// Library/POUs/Additional/MC_SoftSwitchTcp/Structures/SoftSwitchTcpOutCmd
{attribute 'pack_mode' := '1'} 
// ------------------------------------------------------------------------- 
//  SRCI Robot Library                                                
// ------------------------------------------------------------------------- 
//                                                                           
//  Object:      SoftSwitchTcpOutCmd                                       
//  Author:      Thorsten Brach                                                
//  Date:        2024-06-30
//
//  Description:                                              
//   
//                                                                           
//  Copyright: 
//    (C) 2024 Thorsten Brach. All rights reserved                                                                                                                                            
//             Licensed under the LGPL-3.0 license.
//                                                                           
//  Disclaimer:                                                                           
//    This project is provided without any guarantee and can be used for   
//    private and commercial purposes. Any use is at the user’s 
//    own risk and responsibility.
//
// -------------------------------------------------------------------------
TYPE SoftSwitchTcpOutCmd :
STRUCT
  /// If TRUE, the RA is in a compliant movement.
  SoftMovement : BOOL;
END_STRUCT
END_TYPE

// Library/POUs/Additional/MC_SoftSwitchTcp/Structures/SoftSwitchTcpParCmd
{attribute 'pack_mode' := '1'} 
// ------------------------------------------------------------------------- 
//  SRCI Robot Library                                                
// ------------------------------------------------------------------------- 
//                                                                           
//  Object:      SoftSwitchTcpParCmd                                       
//  Author:      Thorsten Brach                                                
//  Date:        2024-06-30
//
//  Description:                                              
//   
//                                                                           
//  Copyright: 
//    (C) 2024 Thorsten Brach. All rights reserved                                                                                                                                            
//             Licensed under the LGPL-3.0 license.
//                                                                           
//  Disclaimer:                                                                           
//    This project is provided without any guarantee and can be used for   
//    private and commercial purposes. Any use is at the user’s 
//    own risk and responsibility.
//
// -------------------------------------------------------------------------
TYPE SoftSwitchTcpParCmd :
STRUCT
  /// Defines type of reference coordinate system at which the robot can be moved in a compliant manner.
  ReferenceType       : ReferenceType;
  /// Index of tool or frame according to ReferenceType.
  /// • 0 (default): Flange/WS
  /// • 1..254: Tool/User frames
  ReferenceNo         : USINT;
  /// Relates to "LimitMode" with the setting "No limit defined". Defines for which cartesian axes the compliant motion is allowed. 
  /// If TRUE, the direction is enabled. Default value is FALSE. See Table 6-744 for bit assignment.
  CompliantAxes       : BYTE;
  /// Defines which parameters will limit the space, where the robot complies (at least one option must be supported)
  LimitMode           : LimitMode;
  /// Defines the type of the resistance force applied at the RA against the external force
  ResistanceForceMode : ResistanceForceMode;
  /// Relates to "ResistanceForceMode" with the setting "ResistanceForceTCP".
  /// Defines the resistance force level applied at the RA against the external force.
  /// • 0..99: Resistance is lower than robot vendor default. The lower the value, the easier the robot can be pushed away.
  /// • 100 (default): The value is aligned with the robot vendor-specific default value.
  /// • 101..200: Resistance is higher than robot vendor default. At maximum value "200" highest possible resistance against external force
  ResistanceForceTCP  : REAL;
  /// Relates to "ResistanceForceMode" with the setting "ResistanceForceAxis".
  /// Defines the resistance force level of the RA at the respective cartesian axis.
  ///  0..99: Resistance is lower than robot vendor default. The lower the value, the easier the robot can be pushed away.
  /// • 100 (default): The value is aligned with the robot vendor-specific default value.
  /// • 101..200: Resistance is higher than robot vendor default. At maximum value "200" highest possible resistance against external force.
  /// Index:
  /// • [0]: X-Axis O
  /// • [1]: Y-axis O
  /// • [2]: Z-axis O
  /// • [3]: RX-Direction O
  /// • [4]: RY-direction O
  /// • [5]: RZ-direction
  ResistanceForceAxis : ARRAY[0..5] OF REAL;
  /// Relates to "LimitMode" with the setting "Limit defined". 
  /// Limit values in the selected cartesian coordinate system (see input parameters ReferenceType and ReferenceNo).
  /// "0" is (default) the origin of the vector, the TCP position, at the start position of the robot.
  /// See Table 6-742 for the parameter index assignment.
  VectorData          : ARRAY[0..5] OF REAL;
END_STRUCT
END_TYPE

// Library/POUs/Additional/MC_SoftSwitchTcp/Structures/SoftSwitchTcpRecvData
{attribute 'pack_mode' := '1'} 
// ------------------------------------------------------------------------- 
//  SRCI Robot Library                                                
// ------------------------------------------------------------------------- 
//                                                                           
//  Object:      SoftSwitchTcpRecvData                                       
//  Author:      Thorsten Brach                                                
//  Date:        2024-06-30
//
//  Description:                                              
//   
//                                                                           
//  Copyright: 
//    (C) 2024 Thorsten Brach. All rights reserved                                                                                                                                            
//             Licensed under the LGPL-3.0 license.
//                                                                           
//  Disclaimer:                                                                           
//    This project is provided without any guarantee and can be used for   
//    private and commercial purposes. Any use is at the user’s 
//    own risk and responsibility.
//
// -------------------------------------------------------------------------
TYPE SoftSwitchTcpRecvData EXTENDS RspHeader :
STRUCT
  /// If TRUE, the RA is in a compliant movement.
  SoftMovement : BOOL;  
END_STRUCT
END_TYPE

// Library/POUs/Additional/MC_SoftSwitchTcp/Structures/SoftSwitchTcpSendData
{attribute 'pack_mode' := '1'}
// ------------------------------------------------------------------------- 
//  SRCI Robot Library                                                
// ------------------------------------------------------------------------- 
//                                                                           
//  Object:      SoftSwitchTcpSendData                                       
//  Author:      Thorsten Brach                                                
//  Date:        2024-06-30
//
//  Description:                                              
//   
//                                                                           
//  Copyright: 
//    (C) 2024 Thorsten Brach. All rights reserved                                                                                                                                            
//             Licensed under the LGPL-3.0 license.
//                                                                           
//  Disclaimer:                                                                           
//    This project is provided without any guarantee and can be used for   
//    private and commercial purposes. Any use is at the user’s 
//    own risk and responsibility.
//
// -------------------------------------------------------------------------
TYPE SoftSwitchTcpSendData EXTENDS CmdHeader: 
STRUCT
  /// Defines which parameters will limit the space, where the robot complies (at least one option must be supported)
  LimitMode           : LimitMode;
  /// Relates to "LimitMode" with the setting "No limit defined". Defines for which cartesian axes the compliant motion is allowed. 
  /// If TRUE, the direction is enabled. Default value is FALSE. See Table 6-744 for bit assignment.
  CompliantAxes       : BYTE;
  /// Defines type of reference coordinate system at which the robot can be moved in a compliant manner.
  ReferenceType       : ReferenceType;  
  /// Index of tool or frame according to ReferenceType.
  /// • 0 (default): Flange/WS
  /// • 1..254: Tool/User frames
  ReferenceNo         : USINT;
  /// Relates to "ResistanceForceMode" with the setting "ResistanceForceTCP".
  /// Defines the resistance force level applied at the RA against the external force.
  /// • 0..99: Resistance is lower than robot vendor default. The lower the value, the easier the robot can be pushed away.
  /// • 100 (default): The value is aligned with the robot vendor-specific default value.
  /// • 101..200: Resistance is higher than robot vendor default. At maximum value "200" highest possible resistance against external force
  ResistanceForceTCP  : INT;
  /// Relates to "ResistanceForceMode" with the setting "ResistanceForceAxis".
  /// Defines the resistance force level of the RA at the respective cartesian axis.
  ///  0..99: Resistance is lower than robot vendor default. The lower the value, the easier the robot can be pushed away.
  /// • 100 (default): The value is aligned with the robot vendor-specific default value.
  /// • 101..200: Resistance is higher than robot vendor default. At maximum value "200" highest possible resistance against external force.
  /// Index:
  /// • [0]: X-Axis O
  /// • [1]: Y-axis O
  /// • [2]: Z-axis O
  /// • [3]: RX-Direction O
  /// • [4]: RY-direction O
  /// • [5]: RZ-direction
  ResistanceForceAxis : ARRAY[0..5] OF UINT;
  /// Relates to "LimitMode" with the setting "Limit defined". 
  /// Limit values in the selected cartesian coordinate system (see input parameters ReferenceType and ReferenceNo).
  /// "0" is (default) the origin of the vector, the TCP position, at the start position of the robot.
  /// See Table 6-742 for the parameter index assignment.
  VectorData          : ARRAY[0..5] OF REAL;
  /// Defines the type of the resistance force applied at the RA against the external force
  ResistanceForceMode : ResistanceForceMode;
END_STRUCT
END_TYPE

// Library/POUs/Additional/MC_StopSubprogram/Structures/StopSubprogramOutCmd
{attribute 'pack_mode' := '1'} 
// ------------------------------------------------------------------------- 
//  SRCI Robot Library                                                
// ------------------------------------------------------------------------- 
//                                                                           
//  Object:      StopSubprogramOutCmd                                       
//  Author:      Thorsten Brach                                                
//  Date:        2024-08-01
//
//  Description:                                              
//   
//                                                                           
//  Copyright: 
//    (C) 2024 Thorsten Brach. All rights reserved                                                                                                                                            
//             Licensed under the LGPL-3.0 license.
//                                                                           
//  Disclaimer:                                                                           
//    This project is provided without any guarantee and can be used for   
//    private and commercial purposes. Any use is at the user’s 
//    own risk and responsibility.
//
// -------------------------------------------------------------------------
TYPE StopSubprogramOutCmd :
STRUCT
  OriginID           : INT;
  /// Relates to ListenerID >0
  /// Number of successful trigger -based command invocations
  /// For more information refer to chapter 5.5.12.4.
  InvocationCounter  : USINT;
END_STRUCT
END_TYPE

// Library/POUs/Additional/MC_StopSubprogram/Structures/StopSubprogramParCmd
{attribute 'pack_mode' := '1'} 
// ------------------------------------------------------------------------- 
//  SRCI Robot Library                                                
// ------------------------------------------------------------------------- 
//                                                                           
//  Object:      StopSubprogramParCmd                                       
//  Author:      Thorsten Brach                                                
//  Date:        2024-08-01
//
//  Description:                                              
//   
//                                                                           
//  Copyright: 
//    (C) 2024 Thorsten Brach. All rights reserved                                                                                                                                            
//             Licensed under the LGPL-3.0 license.
//                                                                           
//  Disclaimer:                                                                           
//    This project is provided without any guarantee and can be used for   
//    private and commercial purposes. Any use is at the user’s 
//    own risk and responsibility.
//
// -------------------------------------------------------------------------
TYPE StopSubprogramParCmd :
STRUCT
  /// Defines how target subprogram is defined
  StopMode          : StopMode;
  /// JobID or InstanceID of target subprogram according to selected StopMode
  /// • Refers to StopMode 0 (Stop via JobID) and 1 (Stop via InstanceID).
  /// • -1: Invalid (default)
  TargetID          : UINT;
  /// Defines the target sequence in which the command will be executed
  SequenceFlag      : SequenceFlag;
  /// ID of associated trigger function:
  /// • 0: No Trigger (default) - No trigger related behavior
  /// • >0: Triggero - Start executing when the trigger function with the identical EmitterID is triggered.
  /// Always positive.
  /// For more information, see chapter 5.5.12 Triggers
  ListenerID        : SINT;
  /// ID of Action that will be executed when this command is active
  /// • >0: Start Action - Start executing the Action function with the identical ListenerID.
  /// • <0: Stop Action  -  Stop executing the Action function with the identical ListenerID.
  /// • 0: No trigger (default)-  If no EmitterID is defined, the function will not trigger any Action during its execution
  /// For more information see section Triggers of this chapter or chapter 5.5.12.4.
  EmitterID          : ARRAY [0..3] OF SINT;  
END_STRUCT
END_TYPE

// Library/POUs/Additional/MC_StopSubprogram/Structures/StopSubprogramRecvData
{attribute 'pack_mode' := '1'} 
// ------------------------------------------------------------------------- 
//  SRCI Robot Library                                                
// ------------------------------------------------------------------------- 
//                                                                           
//  Object:      StopSubprogramRecvData                                       
//  Author:      Thorsten Brach                                                
//  Date:        2024-08-01
//
//  Description:                                              
//   
//                                                                           
//  Copyright: 
//    (C) 2024 Thorsten Brach. All rights reserved                                                                                                                                            
//             Licensed under the LGPL-3.0 license.
//                                                                           
//  Disclaimer:                                                                           
//    This project is provided without any guarantee and can be used for   
//    private and commercial purposes. Any use is at the user’s 
//    own risk and responsibility.
//
// -------------------------------------------------------------------------
TYPE StopSubprogramRecvData EXTENDS RspHeader :
STRUCT
  /// Relates to ListenerID >0
  /// Number of successful trigger-based command invocations - For more information refer TO chapter 5.5.12.4
  InvocationCounter : USINT;  
  /// Reserve
  Reserve           : SINT;
  /// Unique system-generated ID of the "Action" when the function is triggered.
  /// • >0: The "Action" is started by the trigger funcrion with identical FollowID.
  /// • <0: The "Action" is stopped by the trigger function with identical FollowID.
  /// For more information see chapter 5.5.12.4 EmitterID, ListenerID, FollowID and OriginID
  OriginID          : INT;
END_STRUCT
END_TYPE

// Library/POUs/Additional/MC_StopSubprogram/Structures/StopSubprogramSendData
{attribute 'pack_mode' := '1'}
// ------------------------------------------------------------------------- 
//  SRCI Robot Library                                                
// ------------------------------------------------------------------------- 
//                                                                           
//  Object:      StopSubprogramSendData                                       
//  Author:      Thorsten Brach                                                
//  Date:        2024-08-01
//
//  Description:                                              
//   
//                                                                           
//  Copyright: 
//    (C) 2024 Thorsten Brach. All rights reserved                                                                                                                                            
//             Licensed under the LGPL-3.0 license.
//                                                                           
//  Disclaimer:                                                                           
//    This project is provided without any guarantee and can be used for   
//    private and commercial purposes. Any use is at the user’s 
//    own risk and responsibility.
//
// -------------------------------------------------------------------------
TYPE StopSubprogramSendData EXTENDS CmdHeader: 
STRUCT
  /// ID of Action that will be executed when this command is active
  /// • >0: Start Action - Start executing the Action function with the identical ListenerID.
  /// • <0: Stop Action  -  Stop executing the Action function with the identical ListenerID.
  /// • 0: No trigger (default)-  If no EmitterID is defined, the function will not trigger any Action during its execution
  /// For more information see section Triggers of this chapter or chapter 5.5.12.4.
  EmitterID          : ARRAY [0..3] OF SINT;  
  /// ID of associated trigger function:
  /// • 0: No Trigger (default) - No trigger related behavior
  /// • >0: Triggero - Start executing when the trigger function with the identical EmitterID is triggered.
  /// Always positive.
  /// For more information, see chapter 5.5.12 Triggers
  ListenerID        : SINT;
  /// Reserve
  Reserve           : BYTE;
  /// JobID or InstanceID of target subprogram according to selected StopMode
  /// • Refers to StopMode 0 (Stop via JobID) and 1 (Stop via InstanceID).
  /// • -1: Invalid (default)
  TargetID          : UINT;
  /// Defines how target subprogram is defined
  StopMode          : USINT;  
END_STRUCT
END_TYPE

// Library/POUs/Additional/MC_UnitMeasurement/Structures/UnitMeasurementOutCmd
{attribute 'pack_mode' := '1'} 
// ------------------------------------------------------------------------- 
//  SRCI Robot Library                                                
// ------------------------------------------------------------------------- 
//                                                                           
//  Object:      UnitMeasurementOutCmd                                       
//  Author:      Thorsten Brach                                                
//  Date:        2024-06-30
//
//  Description:                                              
//   
//                                                                           
//  Copyright: 
//    (C) 2024 Thorsten Brach. All rights reserved                                                                                                                                            
//             Licensed under the LGPL-3.0 license.
//                                                                           
//  Disclaimer:                                                                           
//    This project is provided without any guarantee and can be used for   
//    private and commercial purposes. Any use is at the user’s 
//    own risk and responsibility.
//
// -------------------------------------------------------------------------
TYPE UnitMeasurementOutCmd :
STRUCT
  /// TRUE, while the measurement is active.
  MeasurementActive : BOOL;
  /// Measurement result depending on the measurement type setting of the "MeasuringMode".
  Result            : REAL;
  /// Unique system-generated ID of the "Action" when the function is triggered.
  /// • >0: The "Action" is started by the trigger function with identical FollowID.
  /// • <0: The "Action" is stopped by the trigger function with identical FollowID.
  /// For more information see chapter 5.5.12.4 EmitterID, ListenerID, FollowID and OriginID
  OriginID           : INT;
  /// Relates to ListenerID >0
  /// Number of successful trigger -based command invocations
  /// For more information refer to chapter 5.5.12.4.
  InvocationCounter  : USINT;
END_STRUCT
END_TYPE

// Library/POUs/Additional/MC_UnitMeasurement/Structures/UnitMeasurementParCmd
{attribute 'pack_mode' := '1'} 
// ------------------------------------------------------------------------- 
//  SRCI Robot Library                                                
// ------------------------------------------------------------------------- 
//                                                                           
//  Object:      UnitMeasurementParCmd                                       
//  Author:      Thorsten Brach                                                
//  Date:        2024-06-30
//
//  Description:                                              
//   
//                                                                           
//  Copyright: 
//    (C) 2024 Thorsten Brach. All rights reserved                                                                                                                                            
//             Licensed under the LGPL-3.0 license.
//                                                                           
//  Disclaimer:                                                                           
//    This project is provided without any guarantee and can be used for   
//    private and commercial purposes. Any use is at the user’s 
//    own risk and responsibility.
//
// -------------------------------------------------------------------------
TYPE UnitMeasurementParCmd :
STRUCT
  ///  Reaction type of measurement in relation to the trigger signal with the "ListenerID > 0" (at least one option must be supported):
  TriggerMode       : TriggerModeMeasurement;
  /// Relates to "TriggerMode" "No trigger related behavior".
  /// Set TRUE to start first measurement. Set TRUE again to receive new result data referring to previous rising edge of NewMeasurement.
  NewMeasurement    : BOOL;  
  /// Type of measurement (at least one option must be supported). 
 /// If the parameter is changed during the active measurement, the RC returns an error
  MeasuringMode     : MeasuringUnitMode;
  /// ID of the trigger function that may be triggered:
  /// • 0: Immediately (default). - Start executing THIS function immediately.
  /// • >0: Triggero Start executing when the trigger function with the identical EmitterID is called.
  /// For more information see chapter 5.5.12.4.
  ListenerID         : SINT;
END_STRUCT
END_TYPE

// Library/POUs/Additional/MC_UnitMeasurement/Structures/UnitMeasurementRecvData
{attribute 'pack_mode' := '1'} 
// ------------------------------------------------------------------------- 
//  SRCI Robot Library                                                
// ------------------------------------------------------------------------- 
//                                                                           
//  Object:      UnitMeasurementRecvData                                       
//  Author:      Thorsten Brach                                                
//  Date:        2024-06-30
//
//  Description:                                              
//   
//                                                                           
//  Copyright: 
//    (C) 2024 Thorsten Brach. All rights reserved                                                                                                                                            
//             Licensed under the LGPL-3.0 license.
//                                                                           
//  Disclaimer:                                                                           
//    This project is provided without any guarantee and can be used for   
//    private and commercial purposes. Any use is at the user’s 
//    own risk and responsibility.
//
// -------------------------------------------------------------------------
TYPE UnitMeasurementRecvData EXTENDS RspHeader :
STRUCT
  /// Relates to ListenerID >0
  /// Number of successful trigger -based command invocations
  /// For more information refer to chapter 5.5.12.4.
  InvocationCounter : USINT;
  /// Reserve
  Reserve           : SINT;
  /// Unique system-generated ID of the "Action" when the function is triggered.
  /// • >0: The "Action" is started by the trigger function with identical FollowID.
  /// • <0: The "Action" is stopped by the trigger function with identical FollowID.
  /// For more information see chapter 5.5.12.4 EmitterID, ListenerID, FollowID and OriginID
  OriginID          : INT;
  /// Measurement result depending on the measurement type setting of the "MeasuringMode".
  Result            : REAL;
  /// TRUE, while the measurement is active.
  MeasurementActive : BOOL;
  /// TRUE, when new result data was received from the RC.
  ResultNo          : USINT;
END_STRUCT
END_TYPE

// Library/POUs/Additional/MC_UnitMeasurement/Structures/UnitMeasurementSendData
{attribute 'pack_mode' := '1'}
// ------------------------------------------------------------------------- 
//  SRCI Robot Library                                                
// ------------------------------------------------------------------------- 
//                                                                           
//  Object:      UnitMeasurementSendData                                       
//  Author:      Thorsten Brach                                                
//  Date:        2024-06-30
//
//  Description:                                              
//   
//                                                                           
//  Copyright: 
//    (C) 2024 Thorsten Brach. All rights reserved                                                                                                                                            
//             Licensed under the LGPL-3.0 license.
//                                                                           
//  Disclaimer:                                                                           
//    This project is provided without any guarantee and can be used for   
//    private and commercial purposes. Any use is at the user’s 
//    own risk and responsibility.
//
// -------------------------------------------------------------------------
TYPE UnitMeasurementSendData EXTENDS CmdHeader: 
STRUCT
  EmitterID     : ARRAY [0..3] OF SINT;
  /// ID of the trigger function that may be triggered:
  /// • 0: Immediately (default). - Start executing THIS function immediately.
  /// • >0: Triggero Start executing when the trigger function with the identical EmitterID is called.
  /// For more information see chapter 5.5.12.4.
  ListenerID    : SINT;
  /// Reserve
  Reserve       : BYTE;
  ///  Reaction type of measurement in relation to the trigger signal with the "ListenerID > 0" (at least one option must be supported):
  TriggerMode   : TriggerModeMeasurement;
  /// Relates to "TriggerMode" "No trigger related behavior".
  /// Set TRUE to start first measurement. Set TRUE again to receive new result data referring to previous rising edge of NewMeasurement.
  MeasurementNo : USINT;
  /// Type of measurement (at least one option must be supported). 
  /// If the parameter is changed during the active measurement, the RC returns an error
  MeasuringMode : MeasuringUnitMode;


END_STRUCT
END_TYPE

// Library/POUs/Additional/MC_WriteCallSubprogramCyclic/Structures/WriteCallSubprogramCyclicOutCmd
{attribute 'pack_mode' := '1'} 
// ------------------------------------------------------------------------- 
//  SRCI Robot Library                                                
// ------------------------------------------------------------------------- 
//                                                                           
//  Object:      UnitMeasurementOutCmd                                       
//  Author:      Thorsten Brach                                                
//  Date:        2024-08-11
//
//  Description:                                              
//   
//                                                                           
//  Copyright: 
//    (C) 2024 Thorsten Brach. All rights reserved                                                                                                                                            
//             Licensed under the LGPL-3.0 license.
//                                                                           
//  Disclaimer:                                                                           
//    This project is provided without any guarantee and can be used for   
//    private and commercial purposes. Any use is at the user’s 
//    own risk and responsibility.
//
// -------------------------------------------------------------------------
TYPE WriteCallSubprogramCyclicOutCmd :
STRUCT

END_STRUCT
END_TYPE

// Library/POUs/Additional/MC_WriteCallSubprogramCyclic/Structures/WriteCallSubprogramCyclicParCmd
{attribute 'pack_mode' := '1'} 
// ------------------------------------------------------------------------- 
//  SRCI Robot Library                                                
// ------------------------------------------------------------------------- 
//                                                                           
//  Object:      UnitMeasurementParCmd                                       
//  Author:      Thorsten Brach                                                
//  Date:        2024-08-11
//
//  Description:                                              
//   
//                                                                           
//  Copyright: 
//    (C) 2024 Thorsten Brach. All rights reserved                                                                                                                                            
//             Licensed under the LGPL-3.0 license.
//                                                                           
//  Disclaimer:                                                                           
//    This project is provided without any guarantee and can be used for   
//    private and commercial purposes. Any use is at the user’s 
//    own risk and responsibility.
//
// -------------------------------------------------------------------------
TYPE WriteCallSubprogramCyclicParCmd :
STRUCT
  /// Cyclic input data of subprogram
  Data : ARRAY[0..25] OF BYTE;
END_STRUCT
END_TYPE

// Library/POUs/AdvancedMove/MC_MoveApproachDirect/Structures/MoveApproachDirectOutCmd
{attribute 'pack_mode' := '1'} 
// ------------------------------------------------------------------------- 
//  SRCI Robot Library                                                
// ------------------------------------------------------------------------- 
//                                                                           
//  Object:      MoveApproachDirectOutCmd                                       
//  Author:      Thorsten Brach                                                
//  Date:        2024-06-30
//
//  Description:                                              
//   
//                                                                           
//  Copyright: 
//    (C) 2024 Thorsten Brach. All rights reserved                                                                                                                                            
//             Licensed under the LGPL-3.0 license.
//                                                                           
//  Disclaimer:                                                                           
//    This project is provided without any guarantee and can be used for   
//    private and commercial purposes. Any use is at the user’s 
//    own risk and responsibility.
//
// -------------------------------------------------------------------------
TYPE MoveApproachDirectOutCmd :
STRUCT
  /// Distance-to-go of the current job.
  /// • -1: No valid value because move command is not yet active (valid values are pending) or not supported by RC
  /// • >0: Actual distance between current and target position
  /// •  0: Target position reached
  RemainingDistance  : REAL;
  /// Percentage of already traversed distance of current job.
  /// If not supported : • -1
  Progress           : REAL;
  /// Unique system-generated ID of the trigger function when the function is called by the user.
  /// For more information see chapter 5.5.12.4.
  FollowID           : DINT;  
END_STRUCT
END_TYPE

// Library/POUs/AdvancedMove/MC_MoveApproachDirect/Structures/MoveApproachDirectParCmd
{attribute 'pack_mode' := '1'} 
// ------------------------------------------------------------------------- 
//  SRCI Robot Library                                                
// ------------------------------------------------------------------------- 
//                                                                           
//  Object:      MoveApproachDirectParCmd                                       
//  Author:      Thorsten Brach                                                
//  Date:        2024-06-30
//
//  Description:                                              
//   
//                                                                           
//  Copyright: 
//    (C) 2024 Thorsten Brach. All rights reserved                                                                                                                                            
//             Licensed under the LGPL-3.0 license.
//                                                                           
//  Disclaimer:                                                                           
//    This project is provided without any guarantee and can be used for   
//    private and commercial purposes. Any use is at the user’s 
//    own risk and responsibility.
//
// -------------------------------------------------------------------------
TYPE MoveApproachDirectParCmd :
STRUCT
  /// Absolute target coordinates in the selected coordinate system (see input parameters ToolNo and FrameNo).
  TargetPosition     : RobotCartesianPosition;
  /// Offset distance of auxiliary position from TargetPosition
  Offset             : AuxOffset;
  /// Defines type of reference coordinate system of the offset position
  ReferenceType      : ReferenceType;
  /// TCP velocity in % of nominal velocity
  /// •  <0%: (default) - Use default velocity
  /// •   0%:           - Use internal minimal velocity
  /// • 100%:           - Use maximal reference velocity
  /// See chapter 5.5.7 Robot dynamics
  VelocityRate       : REAL;
  /// Acceleration for movement in % of nominal acceleration
  /// •  <0%: (default) - Use default acceleration
  /// •   0%:           - Use internal minimal acceleration
  /// • 100%:           - Use maximal reference acceleration
  /// See chapter 5.5.7 Robot dynamics
  AccelerationRate   : REAL;
  /// Deceleration for movement in % of nominal deceleration
  /// •  <0%: (default) - Use default deceleration 
  /// •   0%:           - Use internal minimal deceleration
  /// • 100%:           - Use maximal reference deceleration
  /// See chapter 5.5.7 Robot dynamics
  DecelerationRate   : REAL;
  /// Jerk of the movement in % of nominal jerk
  /// •  <0%: (default) - Use default jerk
  /// •   0%:           - Use internal minimal jerk
  /// • 100%:           - Use maximal reference jerk
  /// See chapter 5.5.7 Robot dynamics
  JerkRate           : REAL;
  /// Index of tool
  /// •      0: Flange (default)
  /// • 1..254: Tool frames
  ToolNo             : USINT;
  /// Index of frame
  /// •      0: WCS (default)
  /// • 1..254: User frames
  FrameNo            : USINT;
  /// Parameter which determines the transition behavior at the end of the movement to be sent to the next command. 
  /// The user can choose a transition type between exact stop and different blend possibilities
  BlendingMode       : BlendingMode;
  /// Additional parameter for the blending mode, to define i.e. velocity limit (%) or blending radius
  BlendingParameter  : ARRAY [0..1] OF REAL := [10,0];
  /// Define blending sphere with radius around auxiliary position. For exact stop define AuxCornerDistance = 0
  AuxCornerDistance  : REAL;
  /// Parameter is used if it is greater than 0 (default)
  /// • Velocity input is ignored
  /// • Parameter defines the time for the movement to reach the target position
  /// Error is sent by the RC if the time cannot be kept
  MoveTime           : TIME;
  /// Parameter to describe how the orientation axes (RX, RY, RZ) will be interpolated during the movement
  OriMode            : OriMode;
  /// Defines the usage of the config byte inside the position according to Table 6-238
  ConfigMode         : ArmConfigParameter;
  /// Defines the usage of the TurnNumber byte inside the position.
  TurnMode           : TurnMode;
  /// Factor by which VelocityRate is multiplied to define the velocity for the second segment of the motion. Always positive.
  /// • 0: use the minimal velocity
  /// • 1: use the velocity set with VelocityRate 
  /// Input values below 1 to reduce velocity, 
  /// Input values above 1 to increase velocity.
  /// See chapter 5.5.7 Robot dynamics
  VelocityCoefficient: REAL;
  /// Set TRUE to allow manipulation of this move command through superimposing functions.
  /// For more information see chapter 5.5.9.5
  Manipulation       : BOOL;
  /// ID of Action that will be executed when this command is active
  /// • >0: Start Action - Start executing the Action function with the identical ListenerID.
  /// • <0: Stop Action  -  Stop executing the Action function with the identical ListenerID.
  /// • 0: No trigger (default)-  If no EmitterID is defined, the function will not trigger any Action during its execution
  /// For more information see section Triggers of this chapter or chapter 5.5.12.4.
  EmitterID          : ARRAY [0..3] OF SINT;
END_STRUCT
END_TYPE

// Library/POUs/AdvancedMove/MC_MoveApproachDirect/Structures/MoveApproachDirectRecvData
{attribute 'pack_mode' := '1'} 
// ------------------------------------------------------------------------- 
//  SRCI Robot Library                                                
// ------------------------------------------------------------------------- 
//                                                                           
//  Object:      MoveApproachDirectRecvData                                       
//  Author:      Thorsten Brach                                                
//  Date:        2024-06-30
//
//  Description:                                              
//   
//                                                                           
//  Copyright: 
//    (C) 2024 Thorsten Brach. All rights reserved                                                                                                                                            
//             Licensed under the LGPL-3.0 license.
//                                                                           
//  Disclaimer:                                                                           
//    This project is provided without any guarantee and can be used for   
//    private and commercial purposes. Any use is at the user’s 
//    own risk and responsibility.
//
// -------------------------------------------------------------------------
TYPE MoveApproachDirectRecvData EXTENDS RspHeader :
STRUCT
  /// Relates to ListenerID >0
  /// Number of successful trigger-based command invocations - For more information refer TO chapter 5.5.12.4
  InvocationCounter : USINT;  
  /// Reserve
  Reserve           : SINT;
  /// Unique system-generated ID of the "Action" when the function is triggered.
  /// • >0: The "Action" is started by the trigger funcrion with identical FollowID.
  /// • <0: The "Action" is stopped by the trigger function with identical FollowID.
  /// For more information see chapter 5.5.12.4 EmitterID, ListenerID, FollowID and OriginID
  OriginID          : INT;
  /// Percentage of already traversed distance of current job.
  /// If not supported : • -1
  Progress          : UINT;
  /// Distance-to-go of the current job.
  /// • -1: No valid value because move command is not yet active (valid values are pending) or not supported by RC
  /// • >0: Actual distance between current and target position
  /// •  0: Target position reached
  RemainingDistance : REAL;
END_STRUCT
END_TYPE

// Library/POUs/AdvancedMove/MC_MoveApproachDirect/Structures/MoveApproachDirectSendData
{attribute 'pack_mode' := '1'}
// ------------------------------------------------------------------------- 
//  SRCI Robot Library                                                
// ------------------------------------------------------------------------- 
//                                                                           
//  Object:      MoveApproachDirectSendData                                       
//  Author:      Thorsten Brach                                                
//  Date:        2024-06-30
//
//  Description:                                              
//   
//                                                                           
//  Copyright: 
//    (C) 2024 Thorsten Brach. All rights reserved                                                                                                                                            
//             Licensed under the LGPL-3.0 license.
//                                                                           
//  Disclaimer:                                                                           
//    This project is provided without any guarantee and can be used for   
//    private and commercial purposes. Any use is at the user’s 
//    own risk and responsibility.
//
// -------------------------------------------------------------------------
TYPE MoveApproachDirectSendData EXTENDS CmdHeader: 
STRUCT
  /// ID of Action that will be executed when this command is active
  /// • >0: Start Action - Start executing the Action function with the identical ListenerID.
  /// • <0: Stop Action  -  Stop executing the Action function with the identical ListenerID.
  /// • 0: No trigger (default)-  If no EmitterID is defined, the function will not trigger any Action during its execution
  /// For more information see section Triggers of this chapter or chapter 5.5.12.4.
  EmitterID          : ARRAY [0..3] OF SINT;
  /// ID of the trigger function that may be triggered:
  /// • 0: Immediately (default). - Start executing THIS function immediately.
  /// • >0: Triggero Start executing when the trigger function with the identical EmitterID is called.
  /// For more information see chapter 5.5.12.4.
  ListenerID         : SINT;
  /// Reserve
  Reserve            : BYTE;
  /// TCP velocity in % of nominal velocity
  /// •  <0%: (default) - Use default velocity
  /// •   0%:           - Use internal minimal velocity
  /// • 100%:           - Use maximal reference velocity
  /// See chapter 5.5.7 Robot dynamics
  VelocityRate       : UINT;  
  /// Acceleration for movement in % of nominal acceleration
  /// •  <0%: (default) - Use default acceleration
  /// •   0%:           - Use internal minimal acceleration
  /// • 100%:           - Use maximal reference acceleration
  /// See chapter 5.5.7 Robot dynamics
  AccelerationRate   : UINT;
  /// Deceleration for movement in % of nominal deceleration
  /// •  <0%: (default) - Use default deceleration 
  /// •   0%:           - Use internal minimal deceleration
  /// • 100%:           - Use maximal reference deceleration
  /// See chapter 5.5.7 Robot dynamics
  DecelerationRate   : UINT;
  /// Jerk of the movement in % of nominal jerk
  /// •  <0%: (default) - Use default jerk
  /// •   0%:           - Use internal minimal jerk
  /// • 100%:           - Use maximal reference jerk
  /// See chapter 5.5.7 Robot dynamics
  JerkRate           : UINT;
  /// Index of tool
  /// •      0: Flange (default)
  /// • 1..254: Tool frames
  ToolNo             : USINT;
  /// Index of frame
  /// •      0: WCS (default)
  /// • 1..254: User frames
  FrameNo            : USINT;
  /// Parameter which determines the transition behavior at the end of the movement to be sent to the next command. 
  /// The user can choose a transition type between exact stop and different blend possibilities
  BlendingMode       : BlendingMode;
  /// Parameter to describe how the orientation axes (RX, RY, RZ) will be interpolated during the movement
  OriMode            : OriMode;
  /// Additional parameter for the blending mode, to define i.e. velocity limit (%) or blending radius
  BlendingParameter  : ARRAY [0..1] OF REAL := [10,0];
  /// Absolute target coordinates in the selected coordinate system (see input parameters ToolNo and FrameNo).
  TargetPosition     : RobotCartesianPosition;
  /// Offset distance of auxiliary position from TargetPosition
  Offset             : AuxOffset;
  /// Define blending sphere with radius around auxiliary position. For exact stop define AuxCornerDistance = 0
  AuxCornerDistance  : REAL;
  /// Factor by which VelocityRate is multiplied to define the velocity for the second segment of the motion. Always positive.
  /// • 0: use the minimal velocity
  /// • 1: use the velocity set with VelocityRate 
  /// Input values below 1 to reduce velocity, 
  /// Input values above 1 to increase velocity.
  /// See chapter 5.5.7 Robot dynamics
  VelocityCoefficient: REAL;
  /// Set TRUE to allow manipulation of this move command through superimposing functions.
  /// For more information see chapter 5.5.9.5
  Manipulation       : BOOL;
  /// Defines the usage of the config byte inside the position according to Table 6-238
  ConfigMode         :  ARRAY[0..1] OF BYTE;
  /// Defines the usage of the TurnNumber byte inside the position.
  TurnMode           : TurnMode;
  /// Defines type of reference coordinate system of the offset position
  ReferenceType      : ReferenceType;
  /// Parameter is used if it is greater than 0 (default)
  /// • Velocity input is ignored
  /// • Parameter defines the time for the movement to reach the target position
  /// Error is sent by the RC if the time cannot be kept
  MoveTime           : UINT;
END_STRUCT
END_TYPE

// Library/POUs/AdvancedMove/MC_MoveApproachLinear/Structures/MoveApproachLinearOutCmd
{attribute 'pack_mode' := '1'} 
// ------------------------------------------------------------------------- 
//  SRCI Robot Library                                                
// ------------------------------------------------------------------------- 
//                                                                           
//  Object:      MoveApproachLinearOutCmd                                       
//  Author:      Thorsten Brach                                                
//  Date:        2024-06-30
//
//  Description:                                              
//   
//                                                                           
//  Copyright: 
//    (C) 2024 Thorsten Brach. All rights reserved                                                                                                                                            
//             Licensed under the LGPL-3.0 license.
//                                                                           
//  Disclaimer:                                                                           
//    This project is provided without any guarantee and can be used for   
//    private and commercial purposes. Any use is at the user’s 
//    own risk and responsibility.
//
// -------------------------------------------------------------------------
TYPE MoveApproachLinearOutCmd :
STRUCT
  /// Distance-to-go of the current job.
  /// • -1: No valid value because move command is not yet active (valid values are pending) or not supported by RC
  /// • >0: Actual distance between current and target position
  /// •  0: Target position reached
  RemainingDistance  : REAL;
  /// Percentage of already traversed distance of current job.
  /// If not supported : • -1
  Progress           : REAL;
  /// Unique system-generated ID of the trigger function when the function is called by the user.
  /// For more information see chapter 5.5.12.4.
  FollowID           : DINT;  
END_STRUCT
END_TYPE

// Library/POUs/AdvancedMove/MC_MoveApproachLinear/Structures/MoveApproachLinearParCmd
{attribute 'pack_mode' := '1'} 
// ------------------------------------------------------------------------- 
//  SRCI Robot Library                                                
// ------------------------------------------------------------------------- 
//                                                                           
//  Object:      MoveApproachLinearParCmd                                       
//  Author:      Thorsten Brach                                                
//  Date:        2024-06-30
//
//  Description:                                              
//   
//                                                                           
//  Copyright: 
//    (C) 2024 Thorsten Brach. All rights reserved                                                                                                                                            
//             Licensed under the LGPL-3.0 license.
//                                                                           
//  Disclaimer:                                                                           
//    This project is provided without any guarantee and can be used for   
//    private and commercial purposes. Any use is at the user’s 
//    own risk and responsibility.
//
// -------------------------------------------------------------------------
TYPE MoveApproachLinearParCmd :
STRUCT
  /// Absolute target coordinates in the selected coordinate system (see input parameters ToolNo and FrameNo).
  TargetPosition     : RobotCartesianPosition;
  /// Offset distance of auxiliary position from TargetPosition
  Offset             : AuxOffset;
  /// Defines type of reference coordinate system of the offset position
  ReferenceType      : ReferenceType;
  /// TCP velocity in % of nominal velocity
  /// •  <0%: (default) - Use default velocity
  /// •   0%:           - Use internal minimal velocity
  /// • 100%:           - Use maximal reference velocity
  /// See chapter 5.5.7 Robot dynamics
  VelocityRate       : REAL;
  /// Acceleration for movement in % of nominal acceleration
  /// •  <0%: (default) - Use default acceleration
  /// •   0%:           - Use internal minimal acceleration
  /// • 100%:           - Use maximal reference acceleration
  /// See chapter 5.5.7 Robot dynamics
  AccelerationRate   : REAL;
  /// Deceleration for movement in % of nominal deceleration
  /// •  <0%: (default) - Use default deceleration 
  /// •   0%:           - Use internal minimal deceleration
  /// • 100%:           - Use maximal reference deceleration
  /// See chapter 5.5.7 Robot dynamics
  DecelerationRate   : REAL;
  /// Jerk of the movement in % of nominal jerk
  /// •  <0%: (default) - Use default jerk
  /// •   0%:           - Use internal minimal jerk
  /// • 100%:           - Use maximal reference jerk
  /// See chapter 5.5.7 Robot dynamics
  JerkRate           : REAL;
  /// Index of tool
  /// •      0: Flange (default)
  /// • 1..254: Tool frames
  ToolNo             : USINT;
  /// Index of frame
  /// •      0: WCS (default)
  /// • 1..254: User frames
  FrameNo            : USINT;
  /// Parameter which determines the transition behavior at the end of the movement to be sent to the next command. 
  /// The user can choose a transition type between exact stop and different blend possibilities
  BlendingMode       : BlendingMode;
  /// Additional parameter for the blending mode, to define i.e. velocity limit (%) or blending radius
  BlendingParameter  : ARRAY [0..1] OF REAL := [10,0];
  /// Define blending sphere with radius around auxiliary position. For exact stop define AuxCornerDistance = 0
  AuxCornerDistance  : REAL;
  /// Parameter is used if it is greater than 0 (default)
  /// • Velocity input is ignored
  /// • Parameter defines the time for the movement to reach the target position
  /// Error is sent by the RC if the time cannot be kept
  MoveTime           : TIME;
  /// Parameter to describe how the orientation axes (RX, RY, RZ) will be interpolated during the movement
  OriMode            : OriMode;
  /// Defines the usage of the config byte inside the position according to Table 6-238
  ConfigMode         : ArmConfigParameter;
  /// Defines the usage of the TurnNumber byte inside the position.
  TurnMode           : TurnMode;
  /// Factor by which VelocityRate is multiplied to define the velocity for the second segment of the motion. Always positive.
  /// • 0: use the minimal velocity
  /// • 1: use the velocity set with VelocityRate 
  /// Input values below 1 to reduce velocity, 
  /// Input values above 1 to increase velocity.
  /// See chapter 5.5.7 Robot dynamics
  VelocityCoefficient: REAL;
  /// Set TRUE to allow manipulation of this move command through superimposing functions.
  /// For more information see chapter 5.5.9.5
  Manipulation       : BOOL;
  /// ID of Action that will be executed when this command is active
  /// • >0: Start Action - Start executing the Action function with the identical ListenerID.
  /// • <0: Stop Action  -  Stop executing the Action function with the identical ListenerID.
  /// • 0: No trigger (default)-  If no EmitterID is defined, the function will not trigger any Action during its execution
  /// For more information see section Triggers of this chapter or chapter 5.5.12.4.
  EmitterID          : ARRAY [0..3] OF SINT;
END_STRUCT
END_TYPE

// Library/POUs/AdvancedMove/MC_MoveApproachLinear/Structures/MoveApproachLinearRecvData
{attribute 'pack_mode' := '1'} 
// ------------------------------------------------------------------------- 
//  SRCI Robot Library                                                
// ------------------------------------------------------------------------- 
//                                                                           
//  Object:      MoveApproachLinearRecvData                                       
//  Author:      Thorsten Brach                                                
//  Date:        2024-06-30
//
//  Description:                                              
//   
//                                                                           
//  Copyright: 
//    (C) 2024 Thorsten Brach. All rights reserved                                                                                                                                            
//             Licensed under the LGPL-3.0 license.
//                                                                           
//  Disclaimer:                                                                           
//    This project is provided without any guarantee and can be used for   
//    private and commercial purposes. Any use is at the user’s 
//    own risk and responsibility.
//
// -------------------------------------------------------------------------
TYPE MoveApproachLinearRecvData EXTENDS RspHeader :
STRUCT
  /// Relates to ListenerID >0
  /// Number of successful trigger-based command invocations - For more information refer TO chapter 5.5.12.4
  InvocationCounter : USINT;  
  /// Reserve
  Reserve           : SINT;
  /// Unique system-generated ID of the "Action" when the function is triggered.
  /// • >0: The "Action" is started by the trigger funcrion with identical FollowID.
  /// • <0: The "Action" is stopped by the trigger function with identical FollowID.
  /// For more information see chapter 5.5.12.4 EmitterID, ListenerID, FollowID and OriginID
  OriginID          : INT;
  /// Percentage of already traversed distance of current job.
  /// If not supported : • -1
  Progress          : UINT;
  /// Distance-to-go of the current job.
  /// • -1: No valid value because move command is not yet active (valid values are pending) or not supported by RC
  /// • >0: Actual distance between current and target position
  /// •  0: Target position reached
  RemainingDistance : REAL;  
END_STRUCT
END_TYPE

// Library/POUs/AdvancedMove/MC_MoveApproachLinear/Structures/MoveApproachLinearSendData
{attribute 'pack_mode' := '1'}
// ------------------------------------------------------------------------- 
//  SRCI Robot Library                                                
// ------------------------------------------------------------------------- 
//                                                                           
//  Object:      MoveApproachLinearSendData                                       
//  Author:      Thorsten Brach                                                
//  Date:        2024-06-30
//
//  Description:                                              
//   
//                                                                           
//  Copyright: 
//    (C) 2024 Thorsten Brach. All rights reserved                                                                                                                                            
//             Licensed under the LGPL-3.0 license.
//                                                                           
//  Disclaimer:                                                                           
//    This project is provided without any guarantee and can be used for   
//    private and commercial purposes. Any use is at the user’s 
//    own risk and responsibility.
//
// -------------------------------------------------------------------------
TYPE MoveApproachLinearSendData EXTENDS CmdHeader: 
STRUCT
/// ID of Action that will be executed when this command is active
  /// • >0: Start Action - Start executing the Action function with the identical ListenerID.
  /// • <0: Stop Action  -  Stop executing the Action function with the identical ListenerID.
  /// • 0: No trigger (default)-  If no EmitterID is defined, the function will not trigger any Action during its execution
  /// For more information see section Triggers of this chapter or chapter 5.5.12.4.
  EmitterID          : ARRAY [0..3] OF SINT;
  /// ID of the trigger function that may be triggered:
  /// • 0: Immediately (default). - Start executing THIS function immediately.
  /// • >0: Triggero Start executing when the trigger function with the identical EmitterID is called.
  /// For more information see chapter 5.5.12.4.
  ListenerID         : SINT;
  /// Reserve
  Reserve            : BYTE;
  /// TCP velocity in % of nominal velocity
  /// •  <0%: (default) - Use default velocity
  /// •   0%:           - Use internal minimal velocity
  /// • 100%:           - Use maximal reference velocity
  /// See chapter 5.5.7 Robot dynamics
  VelocityRate       : UINT;  
  /// Acceleration for movement in % of nominal acceleration
  /// •  <0%: (default) - Use default acceleration
  /// •   0%:           - Use internal minimal acceleration
  /// • 100%:           - Use maximal reference acceleration
  /// See chapter 5.5.7 Robot dynamics
  AccelerationRate   : UINT;
  /// Deceleration for movement in % of nominal deceleration
  /// •  <0%: (default) - Use default deceleration 
  /// •   0%:           - Use internal minimal deceleration
  /// • 100%:           - Use maximal reference deceleration
  /// See chapter 5.5.7 Robot dynamics
  DecelerationRate   : UINT;
  /// Jerk of the movement in % of nominal jerk
  /// •  <0%: (default) - Use default jerk
  /// •   0%:           - Use internal minimal jerk
  /// • 100%:           - Use maximal reference jerk
  /// See chapter 5.5.7 Robot dynamics
  JerkRate           : UINT;
  /// Index of tool
  /// •      0: Flange (default)
  /// • 1..254: Tool frames
  ToolNo             : USINT;
  /// Index of frame
  /// •      0: WCS (default)
  /// • 1..254: User frames
  FrameNo            : USINT;
  /// Parameter which determines the transition behavior at the end of the movement to be sent to the next command. 
  /// The user can choose a transition type between exact stop and different blend possibilities
  BlendingMode       : BlendingMode;
  /// Parameter to describe how the orientation axes (RX, RY, RZ) will be interpolated during the movement
  OriMode            : OriMode;
  /// Additional parameter for the blending mode, to define i.e. velocity limit (%) or blending radius
  BlendingParameter  : ARRAY [0..1] OF REAL := [10,0];
  /// Absolute target coordinates in the selected coordinate system (see input parameters ToolNo and FrameNo).
  TargetPosition     : RobotCartesianPosition;
  /// Offset distance of auxiliary position from TargetPosition
  Offset             : AuxOffset;
  /// Define blending sphere with radius around auxiliary position. For exact stop define AuxCornerDistance = 0
  AuxCornerDistance  : REAL;
  /// Factor by which VelocityRate is multiplied to define the velocity for the second segment of the motion. Always positive.
  /// • 0: use the minimal velocity
  /// • 1: use the velocity set with VelocityRate 
  /// Input values below 1 to reduce velocity, 
  /// Input values above 1 to increase velocity.
  /// See chapter 5.5.7 Robot dynamics
  VelocityCoefficient: REAL;
  /// Set TRUE to allow manipulation of this move command through superimposing functions.
  /// For more information see chapter 5.5.9.5
  Manipulation       : BOOL;
  /// Defines the usage of the config byte inside the position according to Table 6-238
  ConfigMode         :  ARRAY[0..1] OF BYTE;
  /// Defines the usage of the TurnNumber byte inside the position.
  TurnMode           : TurnMode;
  /// Defines type of reference coordinate system of the offset position
  ReferenceType      : ReferenceType;
  /// Parameter is used if it is greater than 0 (default)
  /// • Velocity input is ignored
  /// • Parameter defines the time for the movement to reach the target position
  /// Error is sent by the RC if the time cannot be kept
  MoveTime           : UINT;  
END_STRUCT
END_TYPE

// Library/POUs/AdvancedMove/MC_MoveAxesRelative/Structures/MoveAxesRelativeOutCmd
{attribute 'pack_mode' := '1'} 
// ------------------------------------------------------------------------- 
//  SRCI Robot Library                                                
// ------------------------------------------------------------------------- 
//                                                                           
//  Object:      MoveAxesRelativeOutCmd                                       
//  Author:      Thorsten Brach                                                
//  Date:        2024-07-03
//
//  Description:                                              
//   
//                                                                           
//  Copyright: 
//    (C) 2024 Thorsten Brach. All rights reserved                                                                                                                                            
//             Licensed under the LGPL-3.0 license.
//                                                                           
//  Disclaimer:                                                                           
//    This project is provided without any guarantee and can be used for   
//    private and commercial purposes. Any use is at the user’s 
//    own risk and responsibility.
//
// -------------------------------------------------------------------------
TYPE MoveAxesRelativeOutCmd :
STRUCT
  /// Percentage of already traversed distance of current job.
  /// If not supported : • -1
  Progress           : REAL;
  /// Unique system-generated ID of the trigger function when the function is called by the user.
  /// For more information see chapter 5.5.12.4.
  FollowID           : DINT;
END_STRUCT
END_TYPE

// Library/POUs/AdvancedMove/MC_MoveAxesRelative/Structures/MoveAxesRelativeParCmd
{attribute 'pack_mode' := '1'} 
// ------------------------------------------------------------------------- 
//  SRCI Robot Library                                                
// ------------------------------------------------------------------------- 
//                                                                           
//  Object:      MoveAxesRelativeParCmd                                       
//  Author:      Thorsten Brach                                                
//  Date:        2024-07-03
//
//  Description:                                              
//   
//                                                                           
//  Copyright: 
//    (C) 2024 Thorsten Brach. All rights reserved                                                                                                                                            
//             Licensed under the LGPL-3.0 license.
//                                                                           
//  Disclaimer:                                                                           
//    This project is provided without any guarantee and can be used for   
//    private and commercial purposes. Any use is at the user’s 
//    own risk and responsibility.
//
// -------------------------------------------------------------------------
TYPE MoveAxesRelativeParCmd :
STRUCT
  /// Relative joint distance from the current or last target position to the end joint position
  JointDistance      : RobotJointPosition;
  /// Axes velocity in % of nominal velocity.
  /// •  <0%: (default) - Use default velocity
  /// •   0%:           - Use internal minimal velocity
  /// • 100%:           - Use maximal reference velocity
  /// See chapter 5.5.7 Robot dynamics
  VelocityRate       : REAL;
  /// Acceleration for movement in % of nominal acceleration
  /// •  <0%: (default) - Use default acceleration
  /// •   0%:           - Use internal minimal acceleration
  /// • 100%:           - Use maximal reference acceleration
  /// See chapter 5.5.7 Robot dynamics
  AccelerationRate   : REAL;
  /// Deceleration for movement in % of nominal deceleration
  /// •  <0%: (default) - Use default deceleration 
  /// •   0%:           - Use internal minimal deceleration
  /// • 100%:           - Use maximal reference deceleration
  /// See chapter 5.5.7 Robot dynamics
  DecelerationRate   : REAL;
  /// Jerk of the movement in % of nominal jerk
  /// •  <0%: (default) - Use default jerk
  /// •   0%:           - Use internal minimal jerk
  /// • 100%:           - Use maximal reference jerk
  /// See chapter 5.5.7 Robot dynamics
  JerkRate           : REAL;
  /// Index of tool
  /// •      0: Flange (default)
  /// • 1..254: Tool frames
  ToolNo             : USINT;
  /// Parameter which determines the transition behavior at the end of the movement to be sent to the next command. 
  /// The user can choose a transition type between exact stop and different blend possibilities
  BlendingMode       : BlendingMode;
  /// Additional parameter for the blending mode, to define i.e. velocity limit (%) or blending radius
  BlendingParameter  : ARRAY [0..1] OF REAL := [10,0];
  /// Parameter is used if it is greater than 0 (default)
  /// • Velocity input is ignored
  /// • Parameter defines the time for the movement to reach the target position
  /// Error is sent by the RC if the time cannot be kept
  MoveTime           : TIME;
  /// Set TRUE to allow manipulation of this move command through superimposing functions.
  /// For more information see chapter 5.5.9.5
  Manipulation       : BOOL;
  /// ID of Action that will be executed when this command is active
  /// • >0: Start Action - Start executing the Action function with the identical ListenerID.
  /// • <0: Stop Action  -  Stop executing the Action function with the identical ListenerID.
  /// • 0: No trigger (default)-  If no EmitterID is defined, the function will not trigger any Action during its execution
  /// For more information see section Triggers of this chapter or chapter 5.5.12.4.
  EmitterID          : ARRAY [0..3] OF SINT;
END_STRUCT
END_TYPE

// Library/POUs/AdvancedMove/MC_MoveAxesRelative/Structures/MoveAxesRelativeRecvData
{attribute 'pack_mode' := '1'} 
// ------------------------------------------------------------------------- 
//  SRCI Robot Library                                                
// ------------------------------------------------------------------------- 
//                                                                           
//  Object:      MoveAxesRelativeRecvData                                       
//  Author:      Thorsten Brach                                                
//  Date:        2024-07-03
//
//  Description:                                              
//   
//                                                                           
//  Copyright: 
//    (C) 2024 Thorsten Brach. All rights reserved                                                                                                                                            
//             Licensed under the LGPL-3.0 license.
//                                                                           
//  Disclaimer:                                                                           
//    This project is provided without any guarantee and can be used for   
//    private and commercial purposes. Any use is at the user’s 
//    own risk and responsibility.
//
// -------------------------------------------------------------------------
TYPE MoveAxesRelativeRecvData EXTENDS RspHeader :
STRUCT
  /// Relates to ListenerID >0
  /// Number of successful trigger-based command invocations - For more information refer TO chapter 5.5.12.4
  InvocationCounter : USINT;  
  /// Reserve
  Reserve           : SINT;
  /// Unique system-generated ID of the "Action" when the function is triggered.
  /// • >0: The "Action" is started by the trigger funcrion with identical FollowID.
  /// • <0: The "Action" is stopped by the trigger function with identical FollowID.
  /// For more information see chapter 5.5.12.4 EmitterID, ListenerID, FollowID and OriginID
  OriginID          : INT;
  /// Percentage of already traversed distance of current job.
  /// If not supported : • -1
  Progress          : UINT;
  /// Distance-to-go of the current job.
  /// • -1: No valid value because move command is not yet active (valid values are pending) or not supported by RC
  /// • >0: Actual distance between current and target position
  /// •  0: Target position reached
END_STRUCT
END_TYPE

// Library/POUs/AdvancedMove/MC_MoveAxesRelative/Structures/MoveAxesRelativeSendData
{attribute 'pack_mode' := '1'}
// ------------------------------------------------------------------------- 
//  SRCI Robot Library                                                
// ------------------------------------------------------------------------- 
//                                                                           
//  Object:      MoveAxesRelativeSendData                                       
//  Author:      Thorsten Brach                                                
//  Date:        2024-07-03
//
//  Description:                                              
//   
//                                                                           
//  Copyright: 
//    (C) 2024 Thorsten Brach. All rights reserved                                                                                                                                            
//             Licensed under the LGPL-3.0 license.
//                                                                           
//  Disclaimer:                                                                           
//    This project is provided without any guarantee and can be used for   
//    private and commercial purposes. Any use is at the user’s 
//    own risk and responsibility.
//
// -------------------------------------------------------------------------
TYPE MoveAxesRelativeSendData EXTENDS CmdHeader: 
STRUCT
  /// ID of Action that will be executed when this command is active
  /// • >0: Start Action - Start executing the Action function with the identical ListenerID.
  /// • <0: Stop Action  -  Stop executing the Action function with the identical ListenerID.
  /// • 0: No trigger (default)-  If no EmitterID is defined, the function will not trigger any Action during its execution
  /// For more information see section Triggers of this chapter or chapter 5.5.12.4.
  EmitterID          : ARRAY [0..3] OF SINT;  
  /// ID of the trigger function that may be triggered:
  /// • 0: Immediately (default). - Start executing THIS function immediately.
  /// • >0: Triggero Start executing when the trigger function with the identical EmitterID is called.
  /// For more information see chapter 5.5.12.4.
  ListenerID         : SINT;
  /// Reserve
  Reserve            : SINT;
  /// Axes velocity in % of nominal velocity.
  /// •  <0%: (default) - Use default velocity
  /// •   0%:           - Use internal minimal velocity
  /// • 100%:           - Use maximal reference velocity
  /// See chapter 5.5.7 Robot dynamics
  VelocityRate       : UINT;
  /// Acceleration for movement in % of nominal acceleration
  /// •  <0%: (default) - Use default acceleration
  /// •   0%:           - Use internal minimal acceleration
  /// • 100%:           - Use maximal reference acceleration
  /// See chapter 5.5.7 Robot dynamics
  AccelerationRate   : UINT;
  /// Deceleration for movement in % of nominal deceleration
  /// •  <0%: (default) - Use default deceleration 
  /// •   0%:           - Use internal minimal deceleration
  /// • 100%:           - Use maximal reference deceleration
  /// See chapter 5.5.7 Robot dynamics
  DecelerationRate   : UINT;
  /// Jerk of the movement in % of nominal jerk
  /// •  <0%: (default) - Use default jerk
  /// •   0%:           - Use internal minimal jerk
  /// • 100%:           - Use maximal reference jerk
  /// See chapter 5.5.7 Robot dynamics
  JerkRate           : UINT;
  /// Index of tool
  /// •      0: Flange (default)
  /// • 1..254: Tool frames
  ToolNo             : USINT;
  /// Parameter which determines the transition behavior at the end of the movement to be sent to the next command. 
  /// The user can choose a transition type between exact stop and different blend possibilities
  BlendingMode       : BlendingMode;
  /// Additional parameter for the blending mode, to define i.e. velocity limit (%) or blending radius
  BlendingParameter  : ARRAY [0..1] OF REAL := [10,0];
  /// Relative joint distance from the current or last target position to the end joint position
  JointDistance      : RobotJointPosition;
  /// Set TRUE to allow manipulation of this move command through superimposing functions.
  /// For more information see chapter 5.5.9.5
  Manipulation       : BOOL;
  /// Reserve
  Reserve2           : BYTE;
  /// Parameter is used if it is greater than 0 (default)
  /// • Velocity input is ignored
  /// • Parameter defines the time for the movement to reach the target position
  /// Error is sent by the RC if the time cannot be kept
  MoveTime           : UINT;
END_STRUCT
END_TYPE

// Library/POUs/AdvancedMove/MC_MoveCircularAbsolute/Structures/MoveCircularAbsoluteOutCmd
{attribute 'pack_mode' := '1'} 
// ------------------------------------------------------------------------- 
//  SRCI Robot Library                                                
// ------------------------------------------------------------------------- 
//                                                                           
//  Object:      MoveCircularAbsoluteOutCmd                                       
//  Author:      Thorsten Brach                                                
//  Date:        2024-07-03
//
//  Description:                                              
//   
//                                                                           
//  Copyright: 
//    (C) 2024 Thorsten Brach. All rights reserved                                                                                                                                            
//             Licensed under the LGPL-3.0 license.
//                                                                           
//  Disclaimer:                                                                           
//    This project is provided without any guarantee and can be used for   
//    private and commercial purposes. Any use is at the user’s 
//    own risk and responsibility.
//
// -------------------------------------------------------------------------
TYPE MoveCircularAbsoluteOutCmd :
STRUCT
  /// Distance-to-go of the current job.
  /// • -1: No valid value because move command is not yet active (valid values are pending) or not supported by RC
  /// • >0: Actual distance between current and target position
  /// •  0: Target position reached
  RemainingDistance  : REAL;
  /// Percentage of already traversed distance of current job.
  /// If not supported : • -1
  Progress           : REAL;
  /// Unique system-generated ID of the trigger function when the function is called by the user.
  /// For more information see chapter 5.5.12.4.
  FollowID           : DINT;
END_STRUCT
END_TYPE

// Library/POUs/AdvancedMove/MC_MoveCircularAbsolute/Structures/MoveCircularAbsoluteParCmd
{attribute 'pack_mode' := '1'} 
// ------------------------------------------------------------------------- 
//  SRCI Robot Library                                                
// ------------------------------------------------------------------------- 
//                                                                           
//  Object:      MoveCircularAbsoluteParCmd                                       
//  Author:      Thorsten Brach                                                
//  Date:        2024-07-03
//
//  Description:                                              
//   
//                                                                           
//  Copyright: 
//    (C) 2024 Thorsten Brach. All rights reserved                                                                                                                                            
//             Licensed under the LGPL-3.0 license.
//                                                                           
//  Disclaimer:                                                                           
//    This project is provided without any guarantee and can be used for   
//    private and commercial purposes. Any use is at the user’s 
//    own risk and responsibility.
//
// -------------------------------------------------------------------------
TYPE MoveCircularAbsoluteParCmd :
STRUCT
  /// Specifies the meaning of the input parameter "AuxPoint".
  CircMode           : CircMode;
  /// Auxiliary position of the robot in the specified coordinate system, used in for the circle path calculation.
  AuxPoint           : RobotCartesianPosition;
  /// Specifies the circle’s plane when CircMode = 2 is selected
  CircPlane          : CircPlane;
  /// Relates to CircMode =1:
  /// Permissible deviation of the distances from starting point to center point, from auxiliary point to center point and from end point to center point.
  /// These distances must be identical to travel a circular path. When the distance from a point to the center point is within the allowed deviation, 
  /// the position of the center point is adjusted to the mean internally. If the deviation is greater than the specified Tolerance, 
  /// the command returns an error. See also Figure 6-106.
  Tolerance          : REAL;
  /// Absolute end position of the robot in the specified coordinate system. If "CircMode" = 2 this position is ignored 
  EndPoint           : RobotCartesianPosition;
  /// Angle is only used when "CircMode" = 2. 
  /// The circular angle defines the end position of the circular motion. The circular path is defined by the angle, 
  /// the center point ("AuxPoint") and the actual position. Always positive
  Angle              : REAL;
  /// Choice of the path
  PathChoice         : PathChoice;  
  /// TCP velocity in % of nominal velocity
  /// •  <0%: (default) - Use default velocity
  /// •   0%:           - Use internal minimal velocity
  /// • 100%:           - Use maximal reference velocity
  /// See chapter 5.5.7 Robot dynamics
  VelocityRate       : REAL;
  /// Acceleration for movement in % of nominal acceleration
  /// •  <0%: (default) - Use default acceleration
  /// •   0%:           - Use internal minimal acceleration
  /// • 100%:           - Use maximal reference acceleration
  /// See chapter 5.5.7 Robot dynamics
  AccelerationRate   : REAL;
  /// Deceleration for movement in % of nominal deceleration
  /// •  <0%: (default) - Use default deceleration 
  /// •   0%:           - Use internal minimal deceleration
  /// • 100%:           - Use maximal reference deceleration
  /// See chapter 5.5.7 Robot dynamics
  DecelerationRate   : REAL;
  /// Jerk of the movement in % of nominal jerk
  /// •  <0%: (default) - Use default jerk
  /// •   0%:           - Use internal minimal jerk
  /// • 100%:           - Use maximal reference jerk
  /// See chapter 5.5.7 Robot dynamics
  JerkRate           : REAL;
  /// Index of tool
  /// •      0: Flange (default)
  /// • 1..254: Tool frames
  ToolNo             : USINT;
  /// Index of frame
  /// •      0: WCS (default)
  /// • 1..254: User frames
  FrameNo            : USINT;
  /// Parameter which determines the transition behavior at the end of the movement to be sent to the next command. 
  /// The user can choose a transition type between exact stop and different blend possibilities
  BlendingMode       : BlendingMode;
  /// Additional parameter for the blending mode, to define i.e. velocity limit (%) or blending radius
  BlendingParameter  : ARRAY [0..1] OF REAL := [10,0];
  /// Parameter is used if it is greater than 0 (default)
  /// • Velocity input is ignored
  /// • Parameter defines the time for the movement to reach the target position
  /// Error is sent by the RC if the time cannot be kept
  MoveTime           : TIME;
  /// Parameter to describe how the orientation axes (RX, RY, RZ) will be interpolated during the movement
  OriMode            : OriMode;
  /// Defines the usage of the config byte inside the position according to Table 6-238
  ConfigMode         : ArmConfigParameter;
  /// Defines the usage of the TurnNumber byte inside the position.
  TurnMode           : TurnMode;
  /// Set TRUE to allow manipulation of this move command through superimposing functions.
  /// For more information see chapter 5.5.9.5
  Manipulation       : BOOL;
  /// ID of Action that will be executed when this command is active
  /// • >0: Start Action - Start executing the Action function with the identical ListenerID.
  /// • <0: Stop Action  -  Stop executing the Action function with the identical ListenerID.
  /// • 0: No trigger (default)-  If no EmitterID is defined, the function will not trigger any Action during its execution
  /// For more information see section Triggers of this chapter or chapter 5.5.12.4.
  EmitterID          : ARRAY [0..3] OF SINT;
END_STRUCT
END_TYPE

// Library/POUs/AdvancedMove/MC_MoveCircularAbsolute/Structures/MoveCircularAbsoluteRecvData
{attribute 'pack_mode' := '1'} 
// ------------------------------------------------------------------------- 
//  SRCI Robot Library                                                
// ------------------------------------------------------------------------- 
//                                                                           
//  Object:      MoveCircularAbsoluteRecvData                                       
//  Author:      Thorsten Brach                                                
//  Date:        2024-07-03
//
//  Description:                                              
//   
//                                                                           
//  Copyright: 
//    (C) 2024 Thorsten Brach. All rights reserved                                                                                                                                            
//             Licensed under the LGPL-3.0 license.
//                                                                           
//  Disclaimer:                                                                           
//    This project is provided without any guarantee and can be used for   
//    private and commercial purposes. Any use is at the user’s 
//    own risk and responsibility.
//
// -------------------------------------------------------------------------
TYPE MoveCircularAbsoluteRecvData EXTENDS RspHeader :
STRUCT
  /// Relates to ListenerID >0
  /// Number of successful trigger-based command invocations - For more information refer TO chapter 5.5.12.4
  InvocationCounter : USINT;  
  /// Reserve
  Reserve           : SINT;
  /// Unique system-generated ID of the "Action" when the function is triggered.
  /// • >0: The "Action" is started by the trigger funcrion with identical FollowID.
  /// • <0: The "Action" is stopped by the trigger function with identical FollowID.
  /// For more information see chapter 5.5.12.4 EmitterID, ListenerID, FollowID and OriginID
  OriginID          : INT;
  /// Percentage of already traversed distance of current job.
  /// If not supported : • -1
  Progress          : UINT;
  /// Distance-to-go of the current job.
  /// • -1: No valid value because move command is not yet active (valid values are pending) or not supported by RC
  /// • >0: Actual distance between current and target position
  /// •  0: Target position reached
  RemainingDistance  : REAL;
  
END_STRUCT
END_TYPE

// Library/POUs/AdvancedMove/MC_MoveCircularAbsolute/Structures/MoveCircularAbsoluteSendData
{attribute 'pack_mode' := '1'}
// ------------------------------------------------------------------------- 
//  SRCI Robot Library                                                
// ------------------------------------------------------------------------- 
//                                                                           
//  Object:      MoveCircularAbsoluteSendData                                       
//  Author:      Thorsten Brach                                                
//  Date:        2024-07-03
//
//  Description:                                              
//   
//                                                                           
//  Copyright: 
//    (C) 2024 Thorsten Brach. All rights reserved                                                                                                                                            
//             Licensed under the LGPL-3.0 license.
//                                                                           
//  Disclaimer:                                                                           
//    This project is provided without any guarantee and can be used for   
//    private and commercial purposes. Any use is at the user’s 
//    own risk and responsibility.
//
// -------------------------------------------------------------------------
TYPE MoveCircularAbsoluteSendData EXTENDS CmdHeader: 
STRUCT
  /// ID of Action that will be executed when this command is active
  /// • >0: Start Action - Start executing the Action function with the identical ListenerID.
  /// • <0: Stop Action  -  Stop executing the Action function with the identical ListenerID.
  /// • 0: No trigger (default)-  If no EmitterID is defined, the function will not trigger any Action during its execution
  /// For more information see section Triggers of this chapter or chapter 5.5.12.4.
  EmitterID          : ARRAY [0..3] OF SINT;
  /// ID of the trigger function that may be triggered:
  /// • 0: Immediately (default). - Start executing THIS function immediately.
  /// • >0: Triggero Start executing when the trigger function with the identical EmitterID is called.
  /// For more information see chapter 5.5.12.4.
  ListenerID         : SINT;
  /// Reserve
  Reserve            : SINT;
  /// TCP velocity in % of nominal velocity
  /// •  <0%: (default) - Use default velocity
  /// •   0%:           - Use internal minimal velocity
  /// • 100%:           - Use maximal reference velocity
  /// See chapter 5.5.7 Robot dynamics
  VelocityRate       : UINT;
  /// Acceleration for movement in % of nominal acceleration
  /// •  <0%: (default) - Use default acceleration
  /// •   0%:           - Use internal minimal acceleration
  /// • 100%:           - Use maximal reference acceleration
  /// See chapter 5.5.7 Robot dynamics
  AccelerationRate   : UINT;
  /// Deceleration for movement in % of nominal deceleration
  /// •  <0%: (default) - Use default deceleration 
  /// •   0%:           - Use internal minimal deceleration
  /// • 100%:           - Use maximal reference deceleration
  /// See chapter 5.5.7 Robot dynamics
  DecelerationRate   : UINT;
  /// Jerk of the movement in % of nominal jerk
  /// •  <0%: (default) - Use default jerk
  /// •   0%:           - Use internal minimal jerk
  /// • 100%:           - Use maximal reference jerk
  /// See chapter 5.5.7 Robot dynamics
  JerkRate           : UINT;
  /// Index of tool
  /// •      0: Flange (default)
  /// • 1..254: Tool frames
  ToolNo             : USINT;
  /// Index of frame
  /// •      0: WCS (default)
  /// • 1..254: User frames
  FrameNo            : USINT;
  /// Parameter which determines the transition behavior at the end of the movement to be sent to the next command. 
  /// The user can choose a transition type between exact stop and different blend possibilities
  BlendingMode       : BlendingMode;
  /// Parameter to describe how the orientation axes (RX, RY, RZ) will be interpolated during the movement
  OriMode            : OriMode;
  /// Additional parameter for the blending mode, to define i.e. velocity limit (%) or blending radius
  BlendingParameter  : ARRAY [0..1] OF REAL := [10,0];
  /// Auxiliary position of the robot in the specified coordinate system, used in for the circle path calculation.
  AuxPoint           : RobotCartesianPosition;
  /// Absolute end position of the robot in the specified coordinate system. If "CircMode" = 2 this position is ignored 
  EndPoint           : RobotCartesianPosition;
  /// Specifies the meaning of the input parameter "AuxPoint".
  CircMode           : CircMode;
  /// Specifies the circle’s plane when CircMode = 2 is selected
  CircPlane          : CircPlane;
  /// Relates to CircMode =1:
  /// Permissible deviation of the distances from starting point to center point, from auxiliary point to center point and from end point to center point.
  /// These distances must be identical to travel a circular path. When the distance from a point to the center point is within the allowed deviation, 
  /// the position of the center point is adjusted to the mean internally. If the deviation is greater than the specified Tolerance, 
  /// the command returns an error. See also Figure 6-106.
  Tolerance          : REAL;
  /// Angle is only used when "CircMode" = 2. 
  /// The circular angle defines the end position of the circular motion. The circular path is defined by the angle, 
  /// the center point ("AuxPoint") and the actual position. Always positive
  Angle              : REAL;
  /// Choice of the path
  PathChoice         : bool;  
  /// Set TRUE to allow manipulation of this move command through superimposing functions.
  /// For more information see chapter 5.5.9.5
  Manipulation       : BOOL;
  /// Defines the usage of the config byte inside the position according to Table 6-238
  ConfigMode         : ARRAY[0..1] OF BYTE;
  /// Defines the usage of the TurnNumber byte inside the position.
  TurnMode           : TurnMode;
  /// Reserve
  Reserve2           : BYTE;
  /// Parameter is used if it is greater than 0 (default)
  /// • Velocity input is ignored
  /// • Parameter defines the time for the movement to reach the target position
  /// Error is sent by the RC if the time cannot be kept
  MoveTime           : UINT;
END_STRUCT
END_TYPE

// Library/POUs/AdvancedMove/MC_MoveCircularCamFB/Structures/MoveCircularCamOutCmd
{attribute 'pack_mode' := '1'} 
// ------------------------------------------------------------------------- 
//  SRCI Robot Library                                                
// ------------------------------------------------------------------------- 
//                                                                           
//  Object:      MoveCircularCamOutCmd                                       
//  Author:      Thorsten Brach                                                
//  Date:        2024-07-25
//
//  Description:                                              
//   
//                                                                           
//  Copyright: 
//    (C) 2024 Thorsten Brach. All rights reserved                                                                                                                                            
//             Licensed under the LGPL-3.0 license.
//                                                                           
//  Disclaimer:                                                                           
//    This project is provided without any guarantee and can be used for   
//    private and commercial purposes. Any use is at the user’s 
//    own risk and responsibility.
//
// -------------------------------------------------------------------------
TYPE MoveCircularCamOutCmd :
STRUCT
  /// Percentage of already traversed distance of current job.
  /// If not supported : • -1
  Progress           : REAL;  
  /// Distance-to-go of the current job.
  /// • -1: No valid value because move command is not yet active (valid values are pending) or not supported by RC
  /// • >0: Actual distance between current and target position
  /// •  0: Target position reached
  RemainingDistance  : REAL;  
END_STRUCT
END_TYPE

